{attribute 'qualified_only'}
VAR_GLOBAL
 AI: ARRAY[0..1023] OF BYTE;
END_VAR

(* stored: Version 1.1.0.1, ProductVersion 3.1.4024.5
   GVL AnalogInput: Id {9612c49d-6df7-4e27-8683-015620102242} *)
